FUNCTION_BLOCK F_DEAD_BAND (* Basic Function Block Type *)
  (* Standard: 61499-2 *)
  (* Version 0.0, 2011-08-27, 4DIAC-IDE, 4DIAC-Consortium *)
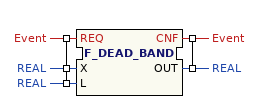
  EVENT_INPUT
    REQ WITH L, X; (* Normal Execution Request *)
  END_EVENT
  EVENT_OUTPUT
    CNF WITH OUT; (* Execution Confirmation *)
  END_EVENT
  VAR_INPUT
    X : REAL; (* input *)
    L : REAL; (* lockout value *)
  END_VAR
  VAR_OUTPUT
    OUT : REAL; (* output *)
  END_VAR
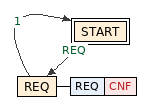
  EC_STATES
    START; (* Initial State *)
    REQ : REQ -> CNF; (* Normal execution *)
  END_STATES
  EC_TRANSITIONS
    START TO REQ := REQ;
    REQ TO START := 1;
  END_TRANSITIONS
  ALGORITHM REQ IN ST: (* Normally executed algorithm *)
IF X > L THEN
	OUT := X - L;
ELSIF X < -L THEN
	OUT := X + L;
ELSE
	OUT := 0.0;
END_IF;
  END_ALGORITHM
END_FUNCTION_BLOCK
